INTERFACE I_EventHandler EXTENDS __SYSTEM.IQueryInterface

METHOD PUBLIC HandleEvent
VAR_INPUT
	Event : I_Event;
END_VAR
END_METHOD

END_INTERFACE

(* stored: Version 1.1.0.1, ProductVersion 3.1.4024.12
   Itf I_EventHandler: Id {56464cbd-e008-4d1d-9019-8281d83ebd69}
   Method HandleEvent: Id {d8fe40f0-d6fe-4487-bf1e-94b1ee695ebe} *)
